// TIA Portal V17 program export: 0 tag tables, 0 data types, 0 data blocks, 3 code blocks (in call order from the OBs), 0 instance data blocks

ORGANIZATION_BLOCK "Main"   // OB1, LAD
BEGIN

REGION Network 1: Call motor control
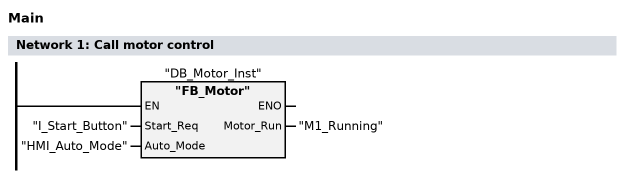
   RUNG wire#powerrail
      "DB_Motor_Inst"(Start_Req := "I_Start_Button", Auto_Mode := "HMI_Auto_Mode", Motor_Run => "M1_Running")
   END_RUNG
   // the same network as SCL:
   "DB_Motor_Inst"(Start_Req := "I_Start_Button", Auto_Mode := "HMI_Auto_Mode", Motor_Run => "M1_Running");   // "FB_Motor"
END_REGION
END_ORGANIZATION_BLOCK

FUNCTION_BLOCK "FB_Motor"   // FB201, LAD
   VAR_INPUT
      Start_Req : Bool;
      Auto_Mode : Bool;
   END_VAR
   VAR_OUTPUT
      Motor_Run : Bool;
   END_VAR
   VAR
      StartDelay : TON_TIME;
   END_VAR
BEGIN

REGION Network 1: Start command interlock
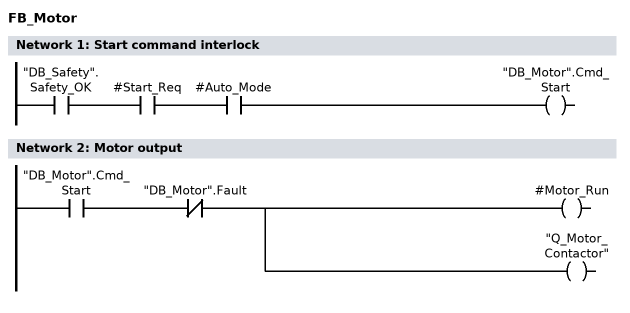
   RUNG wire#powerrail
      Contact( "DB_Safety".Safety_OK )
      Contact( #Start_Req )
      Contact( #Auto_Mode )
      Coil( "DB_Motor".Cmd_Start )
   END_RUNG
   // the same network as SCL:
   "DB_Motor".Cmd_Start := "DB_Safety".Safety_OK AND #Start_Req AND #Auto_Mode;
END_REGION

REGION Network 2: Motor output
   RUNG wire#powerrail
      Contact( "DB_Motor".Cmd_Start )
      I_Contact( "DB_Motor".Fault )
      wire#w1
      Coil( #Motor_Run )
   END_RUNG
   RUNG wire#w1
      Coil( "Q_Motor_Contactor" )
   END_RUNG
   // the same network as SCL:
   #Motor_Run := "DB_Motor".Cmd_Start AND NOT "DB_Motor".Fault;
   "Q_Motor_Contactor" := #Motor_Run;
END_REGION
END_FUNCTION_BLOCK

FUNCTION_BLOCK "FB_Safety"   // FB100, SCL
   VAR_INPUT
      EStop_Ch1 : Bool;
      EStop_Ch2 : Bool;
   END_VAR
BEGIN
// E-Stop evaluation with fault exit
   IF "I_EStop_Button" AND #EStop_Ch1 AND #EStop_Ch2 THEN
       "DB_Safety".Safety_OK := TRUE;
   ELSE
       GOTO FAULT_EXIT;
   END_IF;
   RETURN;
   FAULT_EXIT:
   "DB_Safety".Safety_OK := FALSE;
   "DB_Safety".Fault_Latch := TRUE;
END_FUNCTION_BLOCK
